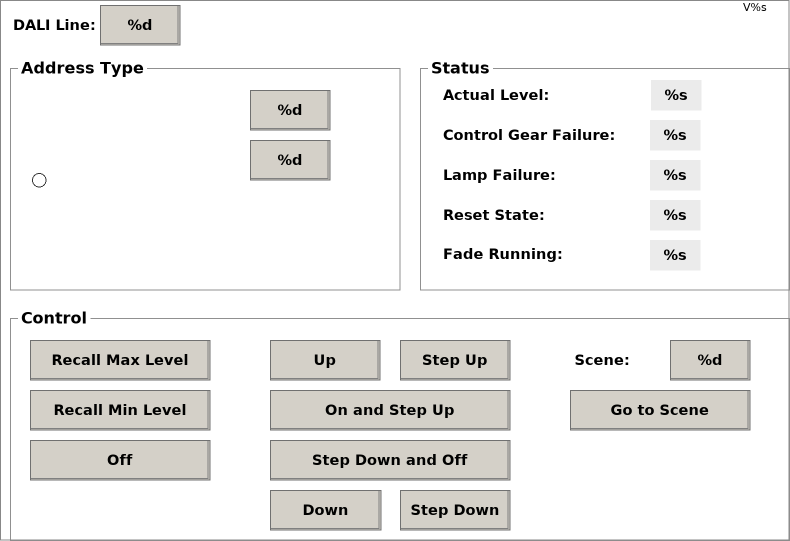
VISUALIZATION Visu_Part102Commands  // 790x541
    GroupBox (10,310 780x231), "Control"
        Button (20,130 180x40), "Off"
            OnMouseClick: execute { DALI_Commissioning.fbPart102Commands.bOff := TRUE; }
        Button (20,80 180x40), "Recall Min Level"
            OnMouseClick: execute { DALI_Commissioning.fbPart102Commands.bRecallMinLevel := TRUE; }
        Button (20,30 180x40), "Recall Max Level"
            OnMouseClick: execute { DALI_Commissioning.fbPart102Commands.bRecallMaxLevel := TRUE; }
        Button (260,180 111x40), "Down"
            OnMouseClick: execute { DALI_Commissioning.fbPart102Commands.bDown := TRUE; }
        Button (390,180 110x40), "Step Down"
            OnMouseClick: execute { DALI_Commissioning.fbPart102Commands.bStepDown := TRUE; }
        Button (260,130 240x40), "Step Down and Off"
            OnMouseClick: execute { DALI_Commissioning.fbPart102Commands.bStepDownAndOff := TRUE; }
        Button (660,30 80x40), "%d", text variable: DALI_Commissioning.fbPart102Commands.nScene
            OnMouseClick: write the text variable via Default, min 0, max 15, title "Insert scene number"
        Textfield (550,35 85x30), "Scene:"
        Button (560,80 180x40), "Go to Scene"
            OnMouseClick: execute { DALI_Commissioning.fbPart102Commands.bGotoScene := TRUE; }
        Button (260,80 240x40), "On and Step Up"
            OnMouseClick: execute { DALI_Commissioning.fbPart102Commands.bOnAndStepUp := TRUE; }
        Button (260,30 110x40), "Up"
            OnMouseClick: execute { DALI_Commissioning.fbPart102Commands.bUp := TRUE; }
        Button (390,30 110x40), "Step Up"
            OnMouseClick: execute { DALI_Commissioning.fbPart102Commands.bStepUp := TRUE; }
    GroupBox (420,60 370x230), "Status"
        Textfield (20,20 200x30), "Actual Level:"
        Textfield (20,60 200x30), "Control Gear Failure:"
        Textfield (231,20 50x30), "%s", text variable: DALI_Commissioning.fbPart102Commands.sActualLevel
        Textfield (230,60 50x30), "%s", text variable: DALI_Commissioning.fbPart102Commands.sControlGearFailure
        Textfield (20,100 200x30), "Lamp Failure:"
        Textfield (230,100 50x30), "%s", text variable: DALI_Commissioning.fbPart102Commands.sLampFailure
        Textfield (20,140 200x30), "Reset State:"
        Textfield (230,140 50x30), "%s", text variable: DALI_Commissioning.fbPart102Commands.sResetState
        Textfield (20,180 200x28), "Fade Running:"
        Textfield (230,180 50x30), "%s", text variable: DALI_Commissioning.fbPart102Commands.sFadeRunning
    GroupBox (10,60 390x230), "Address Type"
        Button (240,30 80x40), "%d", text variable: DALI_Commissioning.fbPart102Commands.nShortAddress
            OnMouseClick: write the text variable via Default, min 0, max 63, title "Insert Short Address"
            OnMouseClick: execute {  }
        RadioButton (20,20 190x200), variable: DALI_Commissioning.fbPart102Commands.eAddressType
            Areas[0]: Text=Short Address
            Areas[1]: Text=Group Address
            Areas[2]: Text=Broadcast
            Areas[3]: Text=Unaddressed
        Button (240,80 80x40), "%d", text variable: DALI_Commissioning.fbPart102Commands.nGroupAddress
            OnMouseClick: write the text variable via Default, min 0, max 15, title "Insert Group Address"
    Rectangle (720,0 70x15), "V%s", text variable: stLibVersion_Tc3_DALI_PLC_Commissioning_Tool.sVersion
    Group (10,5 170x40)
        Textfield (0,0 110x40), "DALI Line:"
        Button (90,0 80x40), "%d", text variable: GVL_Internal.nDALILine
            OnMouseClick: write the text variable via Default, min 1, max 10, title "Choose line"
END_VISUALIZATION

(* stored: Version 1.1.0.1
   Visu Visu_Part102Commands: Id {4f673985-27d9-4ed8-952a-dcd36a46f486} *)
